FUNCTION SubString
VAR_INPUT
	source : ANY;
	destination : ANY;
	startIndex : DINT;
	length : DINT;
END_VAR
VAR
	pTerminator : POINTER TO BYTE;
	numberOfBytes : UDINT;
END_VAR

IF (startIndex >= source.diSize) THEN
	RETURN;
END_IF

numberOfBytes := TO_UDINT(MIN(length, MIN(source.diSize - startIndex, destination.diSize))); 

MEMCPY(
	destAddr := destination.pValue,
	srcAddr := source.pValue + TO_DWORD(startIndex),
	n := numberOfBytes
); 
 
pTerminator := destination.pValue + TO_DWORD(numberOfBytes);
pTerminator^ := 0;

END_FUNCTION

(* stored: Version 1.1.0.1, ProductVersion 3.1.4024.12
   POU SubString: Id {24db83fa-d3af-045a-176e-feaf2ee63db3}, SpecialFunc None *)
